FUNCTION_BLOCK SET_TIMER_DATA (* Sets timer data to machine *)
  (* Standard: 61499-2 *)
  (* Version 1.0, 18-04-2012, GASR, Universidade do Estado de Santa Catarina *)
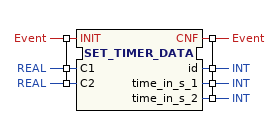
  EVENT_INPUT
    INIT WITH C1, C2;
  END_EVENT
  EVENT_OUTPUT
    CNF WITH id, time_in_s_1, time_in_s_2;
  END_EVENT
  VAR_INPUT
    C1 : REAL; (* Coeficient 1 *)
    C2 : REAL; (* Coeficient 2 *)
  END_VAR
  VAR_OUTPUT
    id : INT;
    time_in_s_1 : INT;
    time_in_s_2 : INT;
  END_VAR
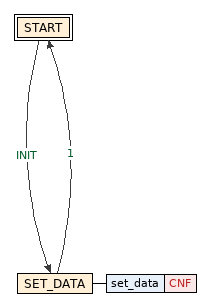
  EC_STATES
    START;
    SET_DATA : set_data -> CNF;
  END_STATES
  EC_TRANSITIONS
    START TO SET_DATA := INIT;
    SET_DATA TO START := 1;
  END_TRANSITIONS
  ALGORITHM set_data IN Lua:
id = C1
local precision = 3
time_in_s_1 = math.floor( C2 )
time_in_s_2 = (C2 - time_in_s_1)*(10^precision)
time_in_s_2 = math.floor( time_in_s_2 )
  END_ALGORITHM
END_FUNCTION_BLOCK
